// Mitsubishi GX Works2 project: 230928-004-PISCA PISCA   PLC: Q03UDV

// task Task_01 (event TRUE, interval 0, priority 31): POU_01

PROGRAM POU_01
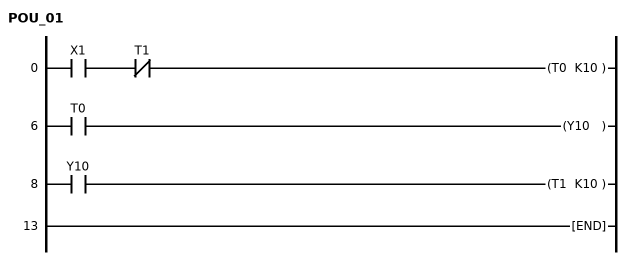
0     LD      X1
      ANI     T1
      OUT     T0 K10
6     LD      T0
      OUT     Y10
8     LD      Y10
      OUT     T1 K10
13    END
END_PROGRAM
